FUNCTION BOOL_BMUX : BOOL
VAR_INPUT
	B: BOOL;
	X: BOOL;
	Y: BOOL
;
END_VAR
VAR
END_VAR

IF NOT B THEN
	BOOL_BMUX := X;
ELSE
	BOOL_BMUX := Y;
END_IF

END_FUNCTION

(* stored: Version 1.1.0.1, ProductVersion 3.1.4024.6
   POU BOOL_BMUX: Id {114651c6-f638-4281-963c-1cdacc01e412}, SpecialFunc None *)
